# EPICS substitutions: iocAdminLib/autosaveSrc/autosave_iocAdmin.substitutions
#
# iocAdmin autosave sample substitutions file
#
file autosave_iocAdmin.template
{
}
